FUNCTION_BLOCK DataProcessing (* Service Interface Function Block Type *)
  (* Standard: 61499-2 *)
  (* Version 1.0, 2023-08-25, ADMIN *)
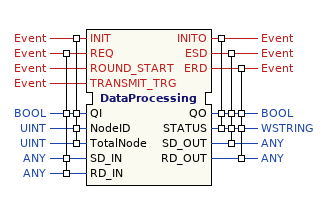
  EVENT_INPUT
    INIT WITH QI, NodeID, TotalNode; (* Service Initialization *)
    REQ WITH QI, SD_IN, RD_IN; (* Service Request *)
    ROUND_START;
    TRANSMIT_TRG;
  END_EVENT
  EVENT_OUTPUT
    INITO WITH QO, STATUS; (* Initialization Confirm *)
    ESD WITH QO, STATUS, SD_OUT; (* Confirmation of Requested Service *)
    ERD WITH RD_OUT, QO, STATUS;
  END_EVENT
  VAR_INPUT
    QI : BOOL; (* Event Input Qualifier *)
    NodeID : UINT; (* Current Node ID *)
    TotalNode : UINT;
    SD_IN : ANY; (* Output data to resource *)
    RD_IN : ANY;
  END_VAR
  VAR_OUTPUT
    QO : BOOL; (* Event Output Qualifier *)
    STATUS : WSTRING; (* Service Status *)
    SD_OUT : ANY; (* Input data from resource *)
    RD_OUT : ANY;
  END_VAR
  (* Service APPLICATION/RESOURCE: Service Interface Function Block Type *)
END_FUNCTION_BLOCK
